Fanuc TP program (LS listing): clskp_g2.ls

/PROG  CLSKP_G2
/ATTR
OWNER		= MNEDITOR;
COMMENT		= "set skip cond g2";
PROG_SIZE	= 320;
CREATE		= DATE 08-10-17  TIME 22:35:26;
MODIFIED	= DATE 08-10-17  TIME 22:36:26;
FILE_NAME	= CLSKP_G1;
VERSION		= 0;
LINE_COUNT	= 6;
MEMORY_SIZE	= 700;
PROTECT		= READ_WRITE;
TCD:  STACK_SIZE	= 0,
      TASK_PRIORITY	= 50,
      TIME_SLICE	= 0,
      BUSY_LAMP_OFF	= 0,
      ABORT_REQUEST	= 0,
      PAUSE_REQUEST	= 0;
DEFAULT_GROUP	= *,*,*,*,*;
CONTROL_CODE	= 00000000 00000000;
/APPL
  SPOT : TRUE ;
/MN
   1:  !Program CLSKP_g2  ;
   2:   ;
   3:  SKIP CONDITION $MISC[2].$DSTB_EXCESS=1    ;
   4:  END ;
   5:   ;
   6:  !End of CLSKP_g2  ;
/POS
/END
